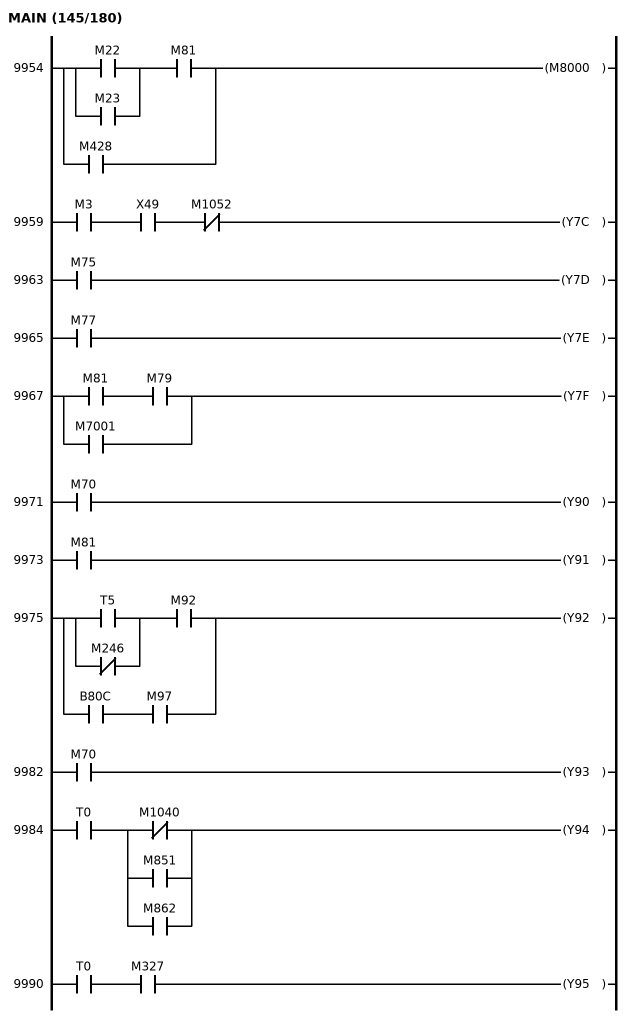
[picture p144: ladder of MAIN, rungs at steps 9954 to 9990]
9954  LD      M22
      OR      M23
      AND     M81
      OR      M428
      OUT     M8000
9959  LD      M3
      AND     X49
      ANI     M1052
      OUT     Y7C
9963  LD      M75
      OUT     Y7D
9965  LD      M77
      OUT     Y7E
9967  LD      M81
      AND     M79
      OR      M7001
      OUT     Y7F
9971  LD      M70
      OUT     Y90
9973  LD      M81
      OUT     Y91
9975  LD      T5
      ORI     M246
      AND     M92
      LD      B80C
      AND     M97
      ORB
      OUT     Y92
9982  LD      M70
      OUT     Y93
9984  LD      T0
      LDI     M1040
      OR      M851
      OR      M862
      ANB
      OUT     Y94
9990  LD      T0
      AND     M327
      OUT     Y95
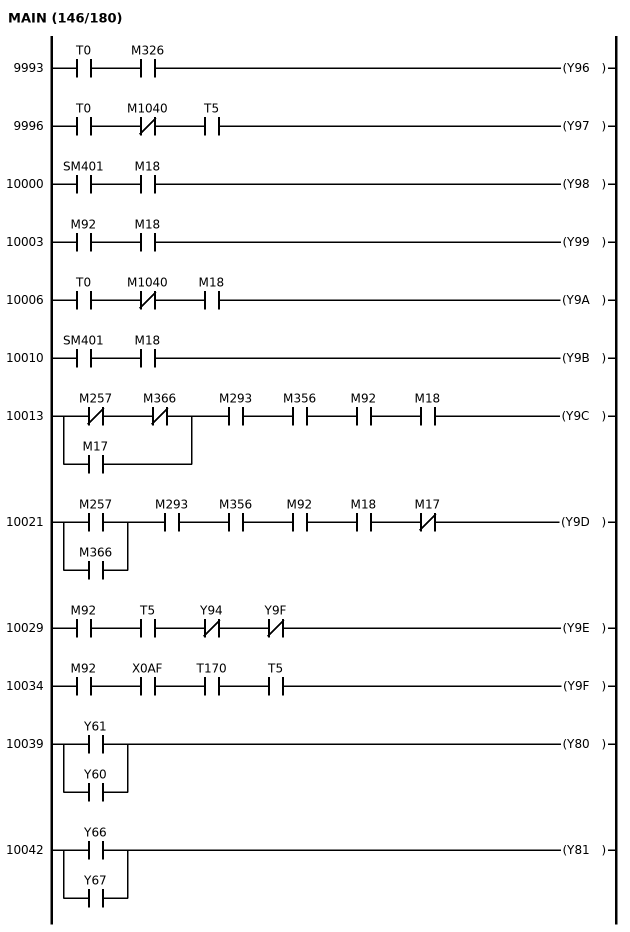
9993  LD      T0
      AND     M326
      OUT     Y96
9996  LD      T0
      ANI     M1040
      AND     T5
      OUT     Y97
10000 LD      SM401
      AND     M18
      OUT     Y98
10003 LD      M92
      AND     M18
      OUT     Y99
10006 LD      T0
      ANI     M1040
      AND     M18
      OUT     Y9A
10010 LD      SM401
      AND     M18
      OUT     Y9B
10013 LDI     M257
      ANI     M366
      OR      M17
      AND     M293
      AND     M356
      AND     M92
      AND     M18
      OUT     Y9C
10021 LD      M257
      OR      M366
      AND     M293
      AND     M356
      AND     M92
      AND     M18
      ANI     M17
      OUT     Y9D
10029 LD      M92
      AND     T5
      ANI     Y94
      ANI     Y9F
      OUT     Y9E
10034 LD      M92
      AND     X0AF
      AND     T170
      AND     T5
      OUT     Y9F
10039 LD      Y61
      OR      Y60
      OUT     Y80
10042 LD      Y66
      OR      Y67
      OUT     Y81
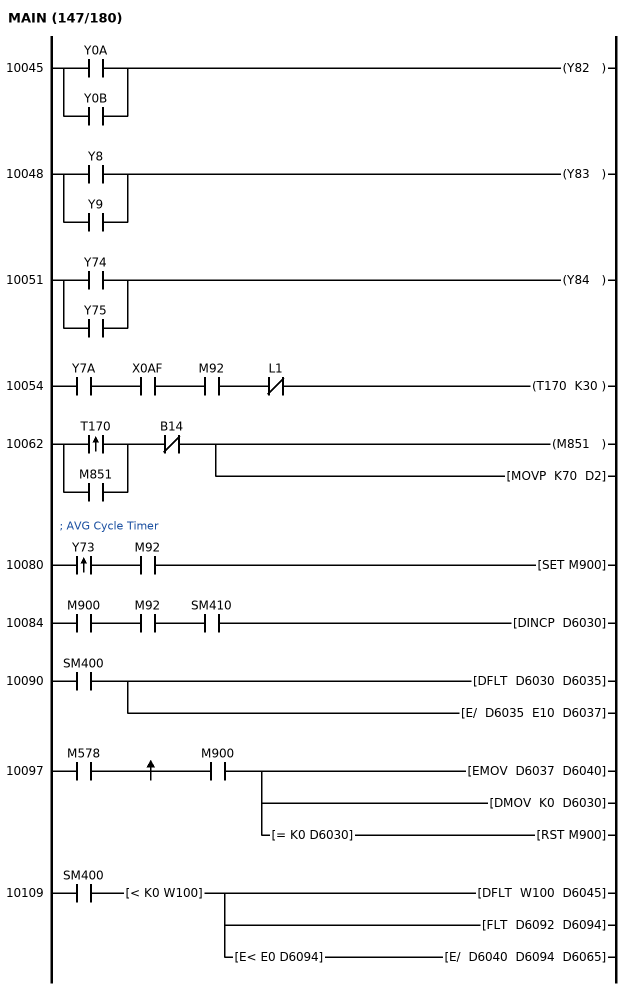
10045 LD      Y0A
      OR      Y0B
      OUT     Y82
10048 LD      Y8
      OR      Y9
      OUT     Y83
10051 LD      Y74
      OR      Y75
      OUT     Y84
10054 LD      Y7A
      AND     X0AF
      AND     M92
      ANI     L1
      OUT     T170 K30
10062 LDP     T170
      OR      M851
      ANI     B14
      OUT     M851
      MOVP    K70 D2
; AVG Cycle Timer
10080 LDP     Y73
      AND     M92
      SET     M900
10084 LD      M900
      AND     M92
      AND     SM410
      DINCP   D6030
10090 LD      SM400
      DFLT    D6030 D6035
      E/      D6035 E10 D6037
10097 LD      M578
      MEP
      AND     M900
      EMOV    D6037 D6040
      DMOV    K0 D6030
      AND=    K0 D6030
      RST     M900
10109 LD      SM400
      AND<    K0 W100
      DFLT    W100 D6045
      FLT     D6092 D6094
      ANDE<   E0 D6094
      E/      D6040 D6094 D6065
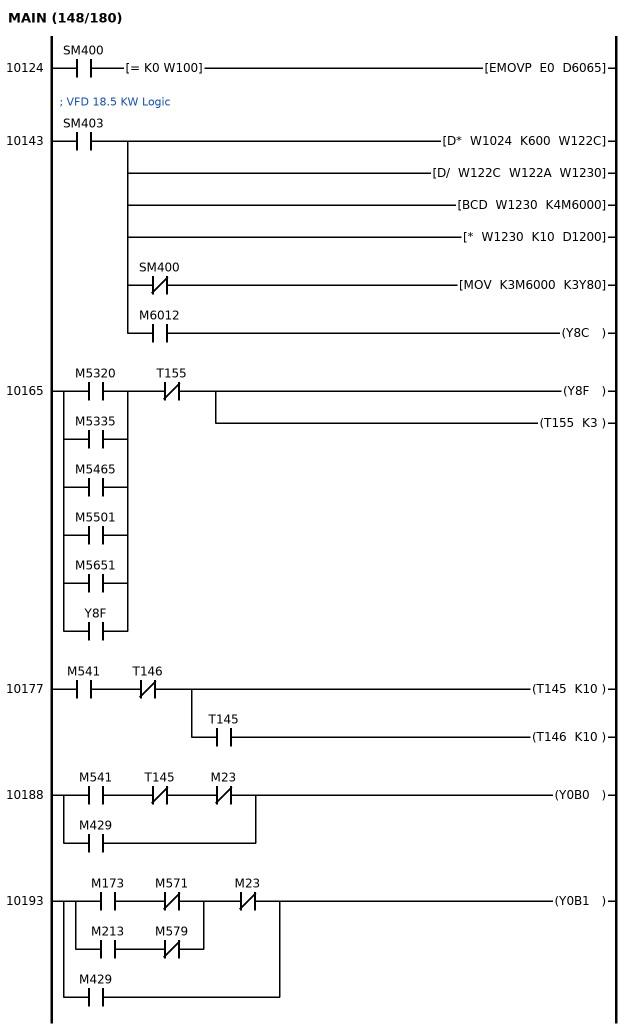
10124 LD      SM400
      AND=    K0 W100
      EMOVP   E0 D6065
; VFD 18.5 KW Logic
10143 LD      SM403
      D*      W1024 K600 W122C
      D/      W122C W122A W1230
      BCD     W1230 K4M6000
      *       W1230 K10 D1200
      MPS
      ANI     SM400
      MOV     K3M6000 K3Y80
      MPP
      AND     M6012
      OUT     Y8C
10165 LD      M5320
      OR      M5335
      OR      M5465
      OR      M5501
      OR      M5651
      OR      Y8F
      ANI     T155
      OUT     Y8F
      OUT     T155 K3
10177 LD      M541
      ANI     T146
      OUT     T145 K10
      AND     T145
      OUT     T146 K10
10188 LD      M541
      ANI     T145
      ANI     M23
      OR      M429
      OUT     Y0B0
10193 LD      M173
      ANI     M571
      LD      M213
      ANI     M579
      ORB
      ANI     M23
      OR      M429
      OUT     Y0B1
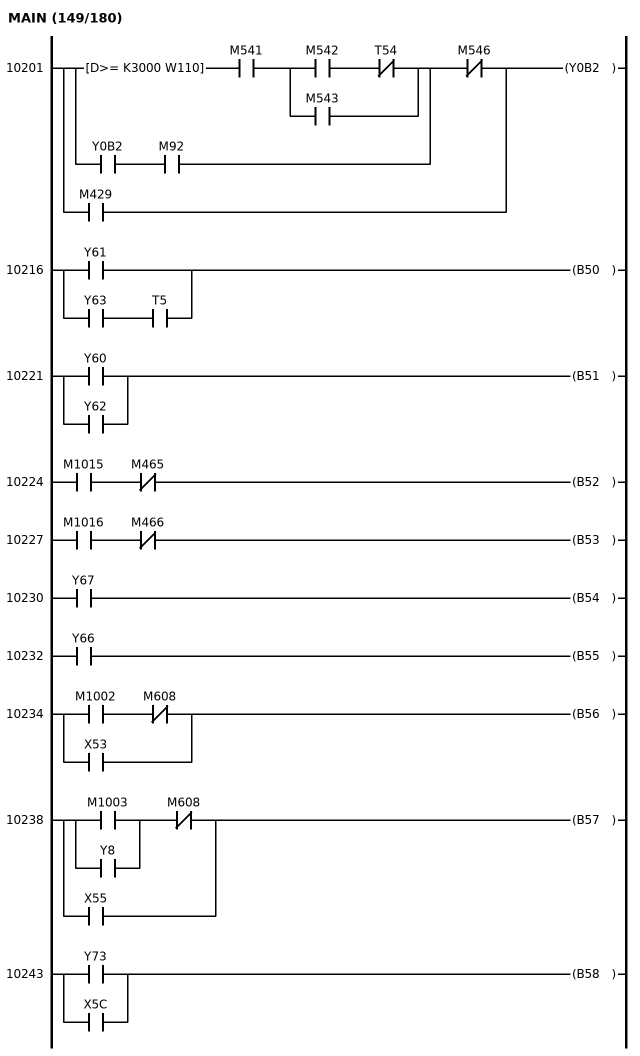
10201 LDD>=   K3000 W110
      AND     M541
      LD      M542
      ANI     T54
      OR      M543
      ANB
      LD      Y0B2
      AND     M92
      ORB
      ANI     M546
      OR      M429
      OUT     Y0B2
10216 LD      Y61
      LD      Y63
      AND     T5
      ORB
      OUT     B50
10221 LD      Y60
      OR      Y62
      OUT     B51
10224 LD      M1015
      ANI     M465
      OUT     B52
10227 LD      M1016
      ANI     M466
      OUT     B53
10230 LD      Y67
      OUT     B54
10232 LD      Y66
      OUT     B55
10234 LD      M1002
      ANI     M608
      OR      X53
      OUT     B56
10238 LD      M1003
      OR      Y8
      ANI     M608
      OR      X55
      OUT     B57
10243 LD      Y73
      OR      X5C
      OUT     B58
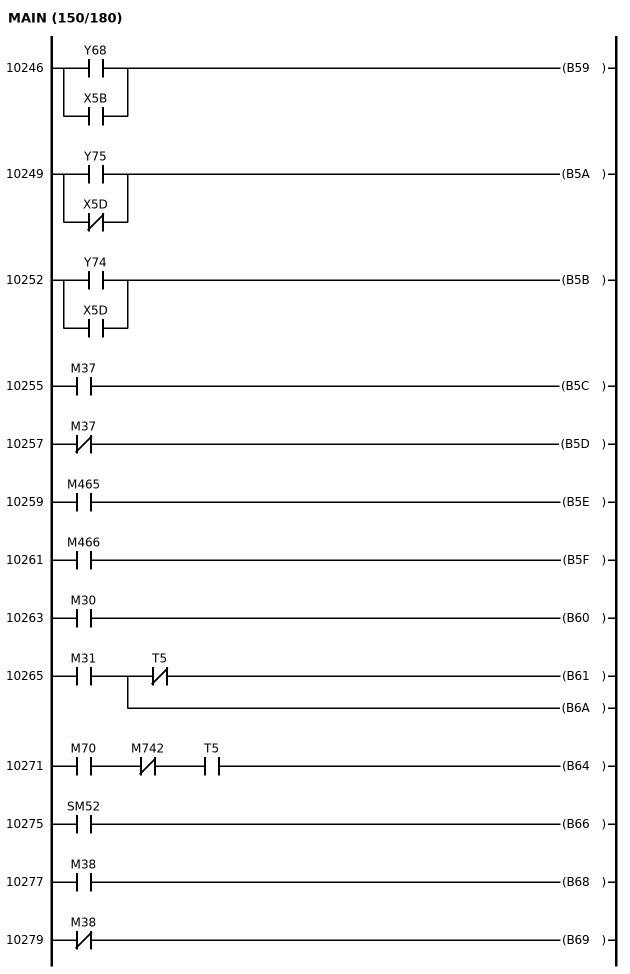
10246 LD      Y68
      OR      X5B
      OUT     B59
10249 LD      Y75
      ORI     X5D
      OUT     B5A
10252 LD      Y74
      OR      X5D
      OUT     B5B
10255 LD      M37
      OUT     B5C
10257 LDI     M37
      OUT     B5D
10259 LD      M465
      OUT     B5E
10261 LD      M466
      OUT     B5F
10263 LD      M30
      OUT     B60
10265 LD      M31
      MPS
      ANI     T5
      OUT     B61
      MPP
      OUT     B6A
10271 LD      M70
      ANI     M742
      AND     T5
      OUT     B64
10275 LD      SM52
      OUT     B66
10277 LD      M38
      OUT     B68
10279 LDI     M38
      OUT     B69
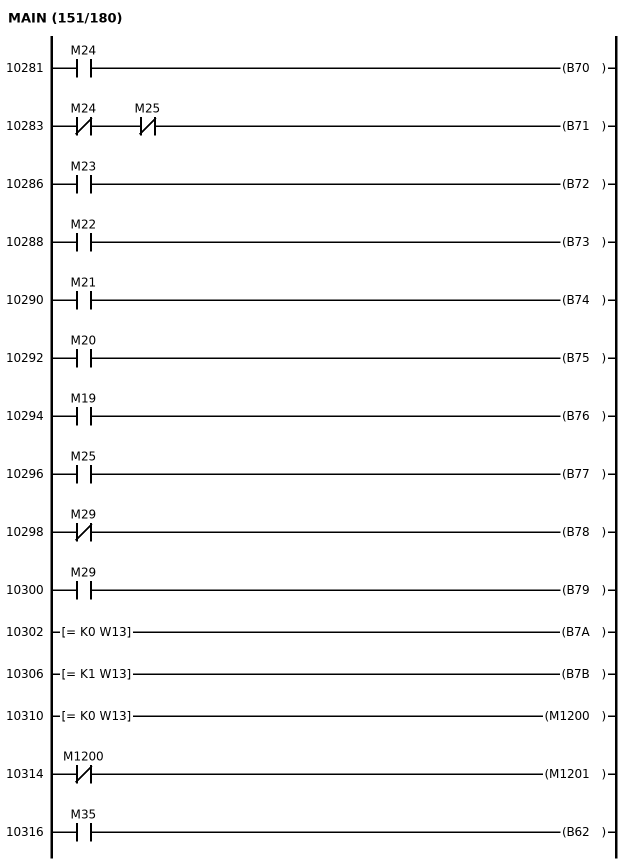
10281 LD      M24
      OUT     B70
10283 LDI     M24
      ANI     M25
      OUT     B71
10286 LD      M23
      OUT     B72
10288 LD      M22
      OUT     B73
10290 LD      M21
      OUT     B74
10292 LD      M20
      OUT     B75
10294 LD      M19
      OUT     B76
10296 LD      M25
      OUT     B77
10298 LDI     M29
      OUT     B78
10300 LD      M29
      OUT     B79
10302 LD=     K0 W13
      OUT     B7A
10306 LD=     K1 W13
      OUT     B7B
10310 LD=     K0 W13
      OUT     M1200
10314 LDI     M1200
      OUT     M1201
10316 LD      M35
      OUT     B62
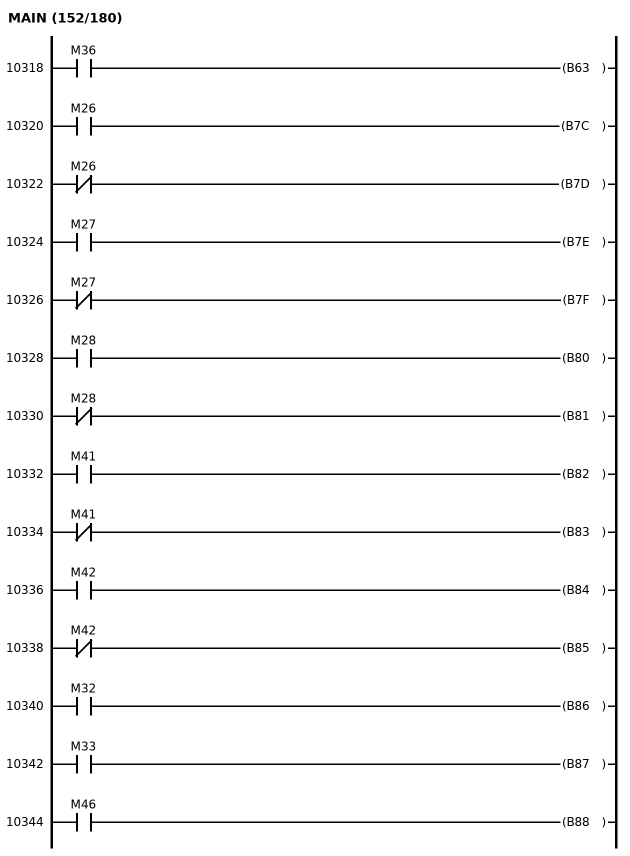
10318 LD      M36
      OUT     B63
10320 LD      M26
      OUT     B7C
10322 LDI     M26
      OUT     B7D
10324 LD      M27
      OUT     B7E
10326 LDI     M27
      OUT     B7F
10328 LD      M28
      OUT     B80
10330 LDI     M28
      OUT     B81
10332 LD      M41
      OUT     B82
10334 LDI     M41
      OUT     B83
10336 LD      M42
      OUT     B84
10338 LDI     M42
      OUT     B85
10340 LD      M32
      OUT     B86
10342 LD      M33
      OUT     B87
10344 LD      M46
      OUT     B88
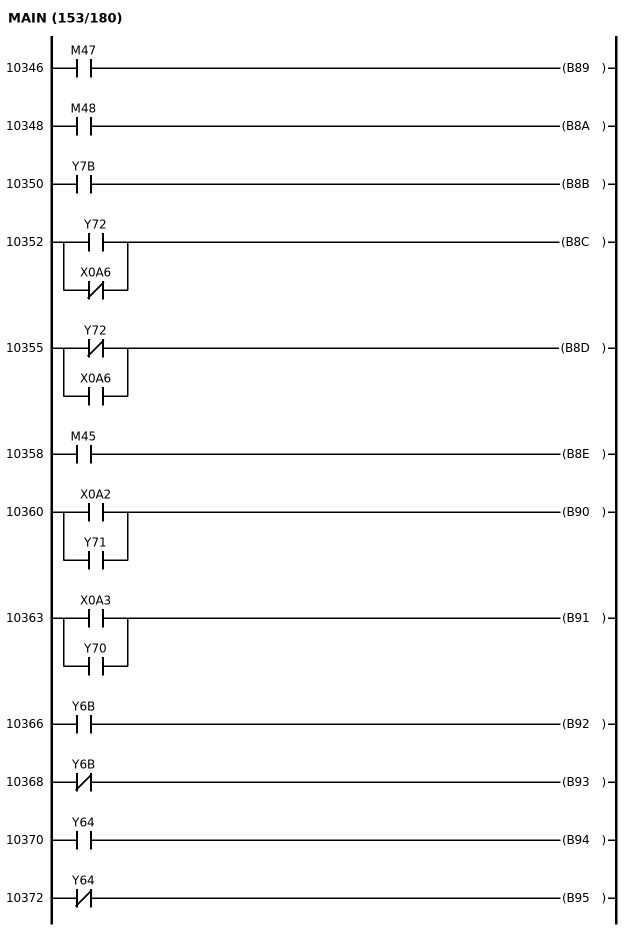
10346 LD      M47
      OUT     B89
10348 LD      M48
      OUT     B8A
10350 LD      Y7B
      OUT     B8B
10352 LD      Y72
      ORI     X0A6
      OUT     B8C
10355 LDI     Y72
      OR      X0A6
      OUT     B8D
10358 LD      M45
      OUT     B8E
10360 LD      X0A2
      OR      Y71
      OUT     B90
10363 LD      X0A3
      OR      Y70
      OUT     B91
10366 LD      Y6B
      OUT     B92
10368 LDI     Y6B
      OUT     B93
10370 LD      Y64
      OUT     B94
10372 LDI     Y64
      OUT     B95
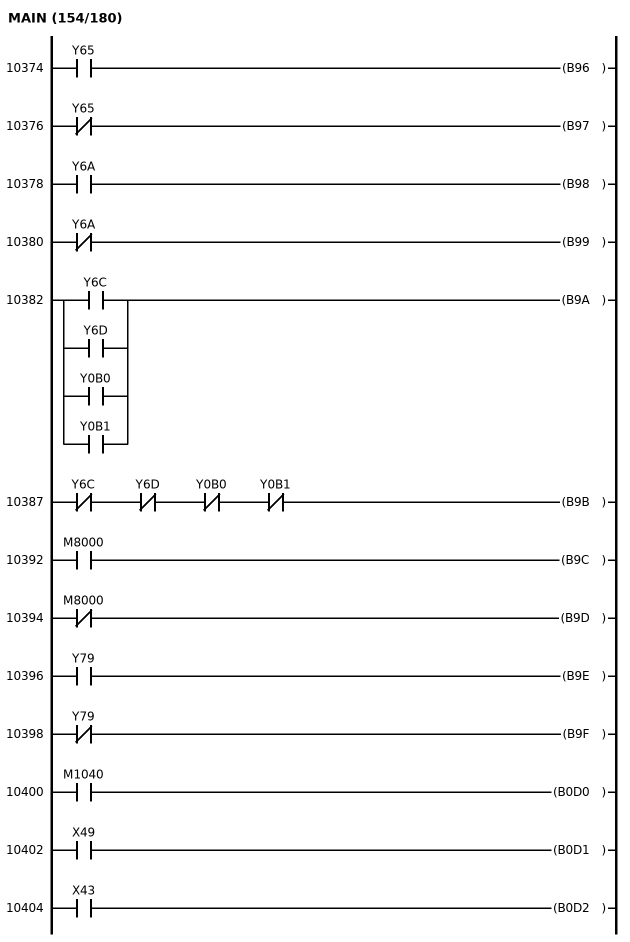
10374 LD      Y65
      OUT     B96
10376 LDI     Y65
      OUT     B97
10378 LD      Y6A
      OUT     B98
10380 LDI     Y6A
      OUT     B99
10382 LD      Y6C
      OR      Y6D
      OR      Y0B0
      OR      Y0B1
      OUT     B9A
10387 LDI     Y6C
      ANI     Y6D
      ANI     Y0B0
      ANI     Y0B1
      OUT     B9B
10392 LD      M8000
      OUT     B9C
10394 LDI     M8000
      OUT     B9D
10396 LD      Y79
      OUT     B9E
10398 LDI     Y79
      OUT     B9F
10400 LD      M1040
      OUT     B0D0
10402 LD      X49
      OUT     B0D1
10404 LD      X43
      OUT     B0D2
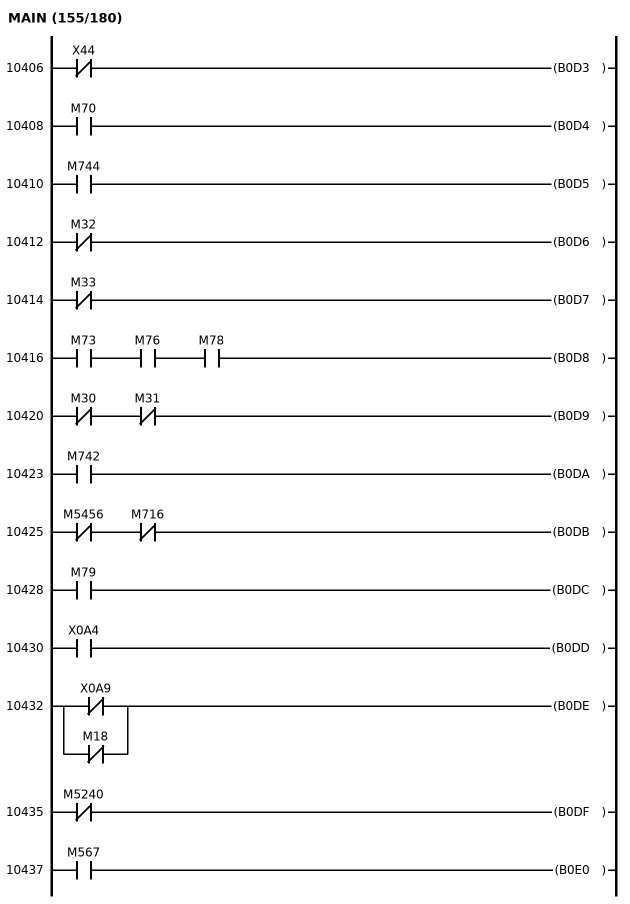
10406 LDI     X44
      OUT     B0D3
10408 LD      M70
      OUT     B0D4
10410 LD      M744
      OUT     B0D5
10412 LDI     M32
      OUT     B0D6
10414 LDI     M33
      OUT     B0D7
10416 LD      M73
      AND     M76
      AND     M78
      OUT     B0D8
10420 LDI     M30
      ANI     M31
      OUT     B0D9
10423 LD      M742
      OUT     B0DA
10425 LDI     M5456
      ANI     M716
      OUT     B0DB
10428 LD      M79
      OUT     B0DC
10430 LD      X0A4
      OUT     B0DD
10432 LDI     X0A9
      ORI     M18
      OUT     B0DE
10435 LDI     M5240
      OUT     B0DF
10437 LD      M567
      OUT     B0E0
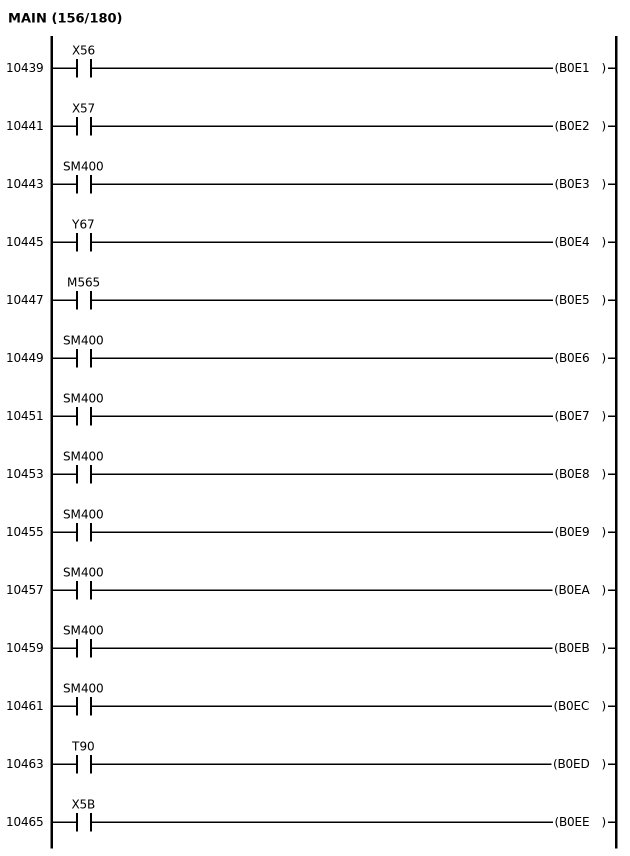
10439 LD      X56
      OUT     B0E1
10441 LD      X57
      OUT     B0E2
10443 LD      SM400
      OUT     B0E3
10445 LD      Y67
      OUT     B0E4
10447 LD      M565
      OUT     B0E5
10449 LD      SM400
      OUT     B0E6
10451 LD      SM400
      OUT     B0E7
10453 LD      SM400
      OUT     B0E8
10455 LD      SM400
      OUT     B0E9
10457 LD      SM400
      OUT     B0EA
10459 LD      SM400
      OUT     B0EB
10461 LD      SM400
      OUT     B0EC
10463 LD      T90
      OUT     B0ED
10465 LD      X5B
      OUT     B0EE
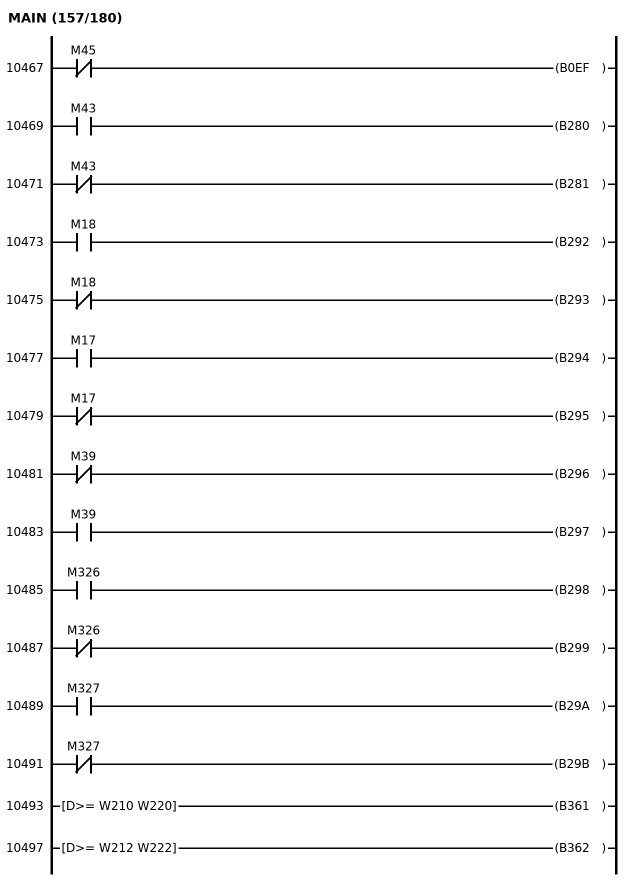
10467 LDI     M45
      OUT     B0EF
10469 LD      M43
      OUT     B280
10471 LDI     M43
      OUT     B281
10473 LD      M18
      OUT     B292
10475 LDI     M18
      OUT     B293
10477 LD      M17
      OUT     B294
10479 LDI     M17
      OUT     B295
10481 LDI     M39
      OUT     B296
10483 LD      M39
      OUT     B297
10485 LD      M326
      OUT     B298
10487 LDI     M326
      OUT     B299
10489 LD      M327
      OUT     B29A
10491 LDI     M327
      OUT     B29B
10493 LDD>=   W210 W220
      OUT     B361
10497 LDD>=   W212 W222
      OUT     B362
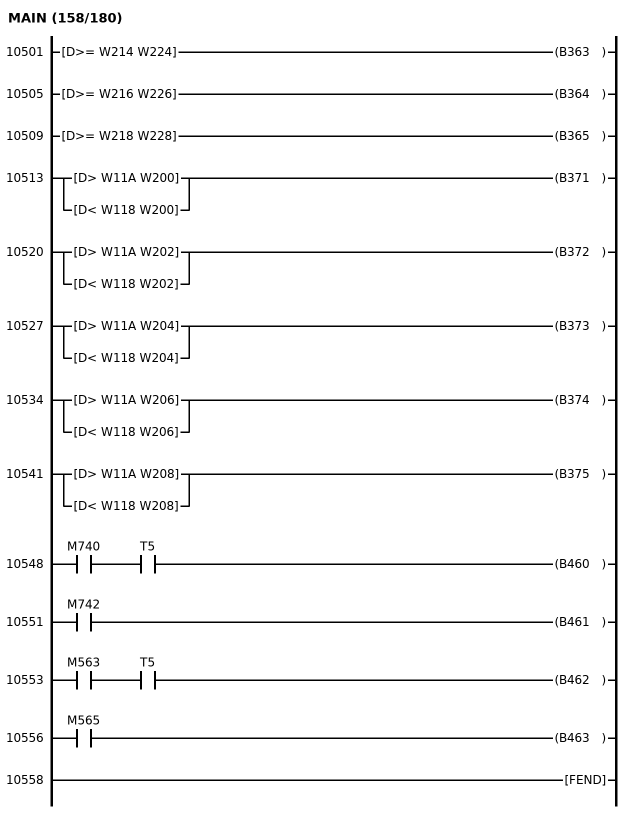
10501 LDD>=   W214 W224
      OUT     B363
10505 LDD>=   W216 W226
      OUT     B364
10509 LDD>=   W218 W228
      OUT     B365
10513 LDD>    W11A W200
      ORD<    W118 W200
      OUT     B371
10520 LDD>    W11A W202
      ORD<    W118 W202
      OUT     B372
10527 LDD>    W11A W204
      ORD<    W118 W204
      OUT     B373
10534 LDD>    W11A W206
      ORD<    W118 W206
      OUT     B374
10541 LDD>    W11A W208
      ORD<    W118 W208
      OUT     B375
10548 LD      M740
      AND     T5
      OUT     B460
10551 LD      M742
      OUT     B461
10553 LD      M563
      AND     T5
      OUT     B462
10556 LD      M565
      OUT     B463
10558 FEND
      P0
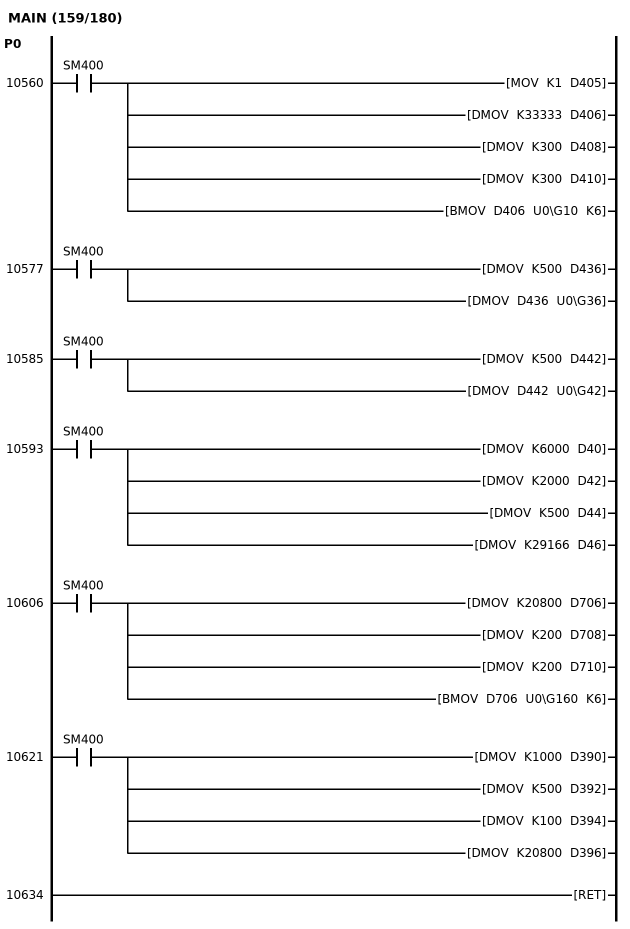
10560 LD      SM400
      MOV     K1 D405
      DMOV    K33333 D406
      DMOV    K300 D408
      DMOV    K300 D410
      BMOV    D406 U0\G10 K6
10577 LD      SM400
      DMOV    K500 D436
      DMOV    D436 U0\G36
10585 LD      SM400
      DMOV    K500 D442
      DMOV    D442 U0\G42
10593 LD      SM400
      DMOV    K6000 D40
      DMOV    K2000 D42
      DMOV    K500 D44
      DMOV    K29166 D46
10606 LD      SM400
      DMOV    K20800 D706
      DMOV    K200 D708
      DMOV    K200 D710
      BMOV    D706 U0\G160 K6
10621 LD      SM400
      DMOV    K1000 D390
      DMOV    K500 D392
      DMOV    K100 D394
      DMOV    K20800 D396
10634 RET
      P1
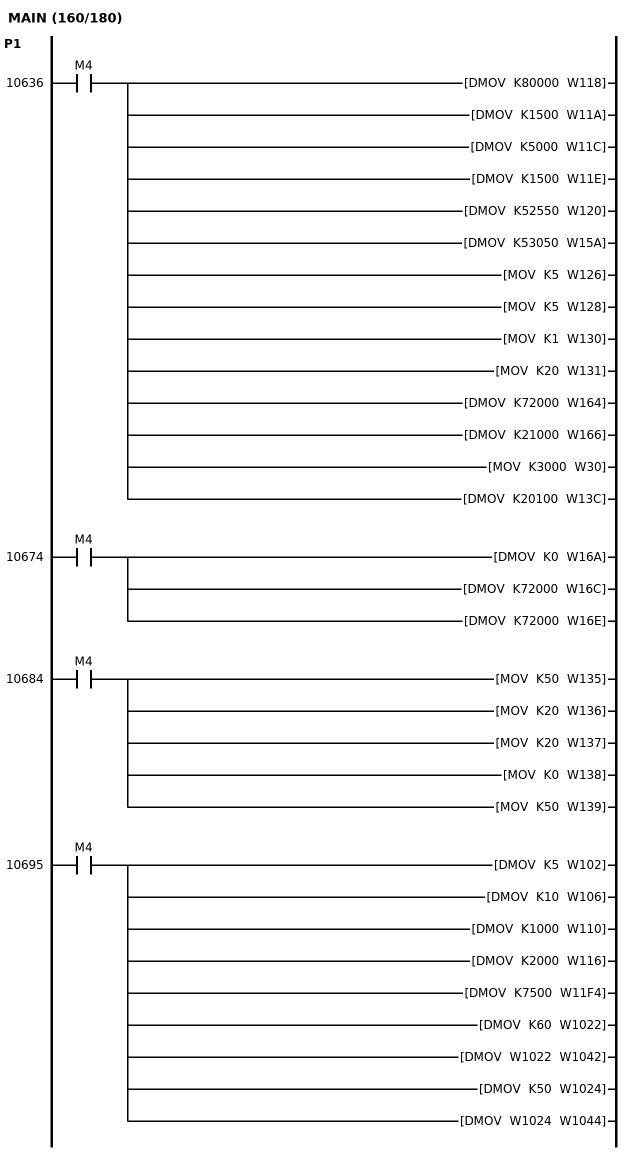
10636 LD      M4
      DMOV    K80000 W118
      DMOV    K1500 W11A
      DMOV    K5000 W11C
      DMOV    K1500 W11E
      DMOV    K52550 W120
      DMOV    K53050 W15A
      MOV     K5 W126
      MOV     K5 W128
      MOV     K1 W130
      MOV     K20 W131
      DMOV    K72000 W164
      DMOV    K21000 W166
      MOV     K3000 W30
      DMOV    K20100 W13C
10674 LD      M4
      DMOV    K0 W16A
      DMOV    K72000 W16C
      DMOV    K72000 W16E
10684 LD      M4
      MOV     K50 W135
      MOV     K20 W136
      MOV     K20 W137
      MOV     K0 W138
      MOV     K50 W139
10695 LD      M4
      DMOV    K5 W102
      DMOV    K10 W106
      DMOV    K1000 W110
      DMOV    K2000 W116
      DMOV    K7500 W11F4
      DMOV    K60 W1022
      DMOV    W1022 W1042
      DMOV    K50 W1024
      DMOV    W1024 W1044
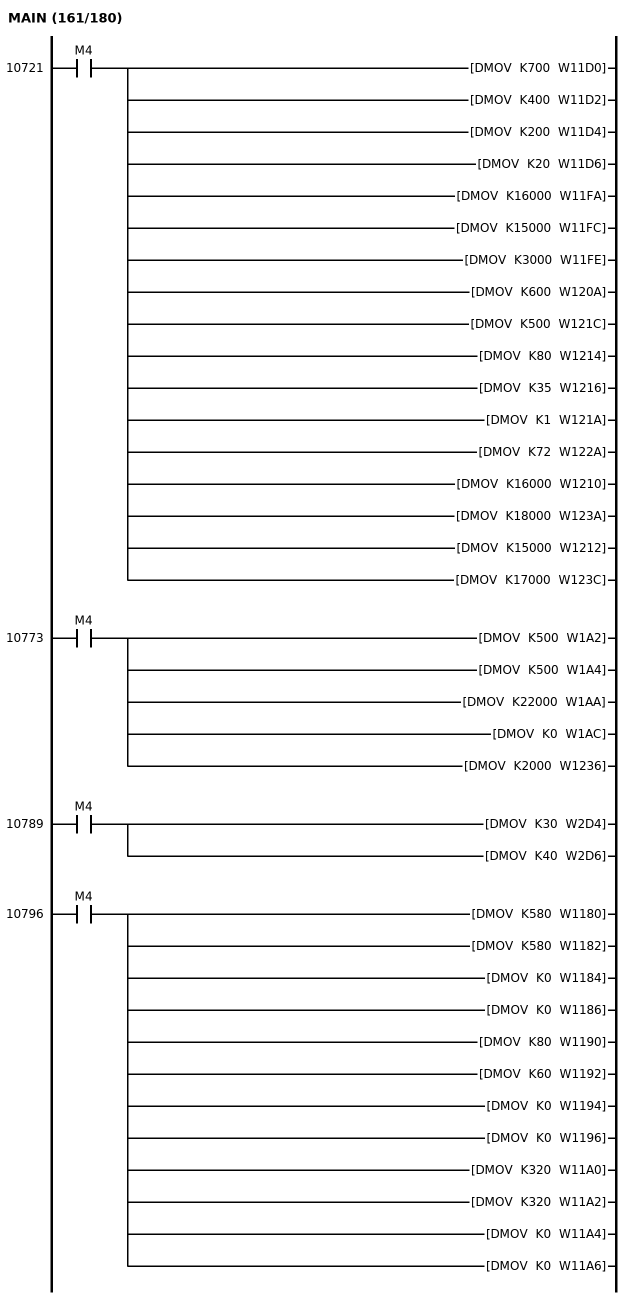
10721 LD      M4
      DMOV    K700 W11D0
      DMOV    K400 W11D2
      DMOV    K200 W11D4
      DMOV    K20 W11D6
      DMOV    K16000 W11FA
      DMOV    K15000 W11FC
      DMOV    K3000 W11FE
      DMOV    K600 W120A
      DMOV    K500 W121C
      DMOV    K80 W1214
      DMOV    K35 W1216
      DMOV    K1 W121A
      DMOV    K72 W122A
      DMOV    K16000 W1210
      DMOV    K18000 W123A
      DMOV    K15000 W1212
      DMOV    K17000 W123C
10773 LD      M4
      DMOV    K500 W1A2
      DMOV    K500 W1A4
      DMOV    K22000 W1AA
      DMOV    K0 W1AC
      DMOV    K2000 W1236
10789 LD      M4
      DMOV    K30 W2D4
      DMOV    K40 W2D6
10796 LD      M4
      DMOV    K580 W1180
      DMOV    K580 W1182
      DMOV    K0 W1184
      DMOV    K0 W1186
      DMOV    K80 W1190
      DMOV    K60 W1192
      DMOV    K0 W1194
      DMOV    K0 W1196
      DMOV    K320 W11A0
      DMOV    K320 W11A2
      DMOV    K0 W11A4
      DMOV    K0 W11A6
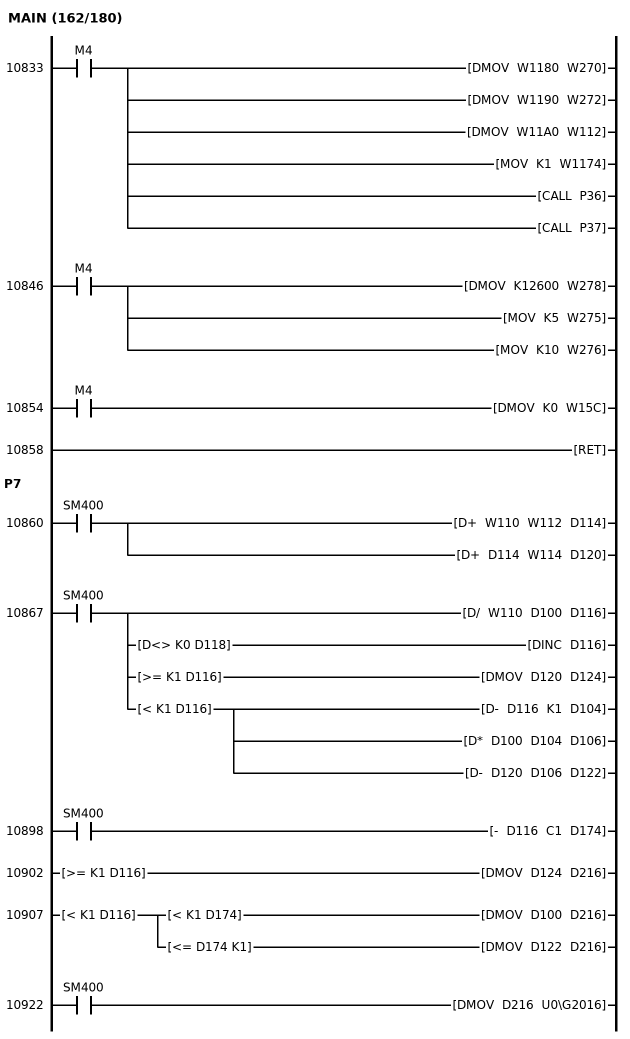
10833 LD      M4
      DMOV    W1180 W270
      DMOV    W1190 W272
      DMOV    W11A0 W112
      MOV     K1 W1174
      CALL    P36
      CALL    P37
10846 LD      M4
      DMOV    K12600 W278
      MOV     K5 W275
      MOV     K10 W276
10854 LD      M4
      DMOV    K0 W15C
10858 RET
      P7
10860 LD      SM400
      D+      W110 W112 D114
      D+      D114 W114 D120
10867 LD      SM400
      D/      W110 D100 D116
      MPS
      ANDD<>  K0 D118
      DINC    D116
      MRD
      AND>=   K1 D116
      DMOV    D120 D124
      MPP
      AND<    K1 D116
      D-      D116 K1 D104
      D*      D100 D104 D106
      D-      D120 D106 D122
10898 LD      SM400
      -       D116 C1 D174
10902 LD>=    K1 D116
      DMOV    D124 D216
10907 LD<     K1 D116
      MPS
      AND<    K1 D174
      DMOV    D100 D216
      MPP
      AND<=   D174 K1
      DMOV    D122 D216
10922 LD      SM400
      DMOV    D216 U0\G2016
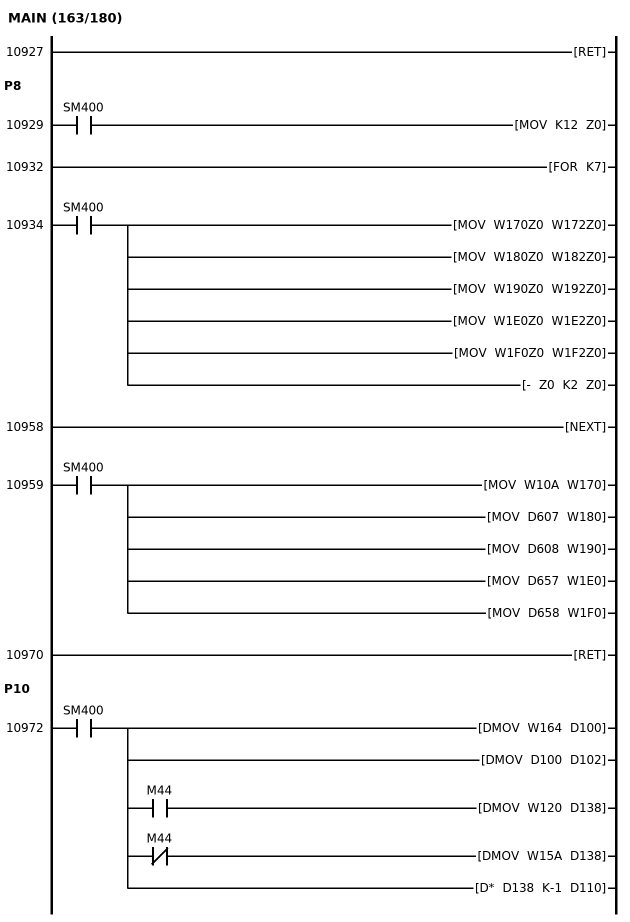
10927 RET
      P8
10929 LD      SM400
      MOV     K12 Z0
10932 FOR     K7
10934 LD      SM400
      MOV     W170Z0 W172Z0
      MOV     W180Z0 W182Z0
      MOV     W190Z0 W192Z0
      MOV     W1E0Z0 W1E2Z0
      MOV     W1F0Z0 W1F2Z0
      -       Z0 K2 Z0
10958 NEXT
10959 LD      SM400
      MOV     W10A W170
      MOV     D607 W180
      MOV     D608 W190
      MOV     D657 W1E0
      MOV     D658 W1F0
10970 RET
      P10
10972 LD      SM400
      DMOV    W164 D100
      DMOV    D100 D102
      MPS
      AND     M44
      DMOV    W120 D138
      MRD
      ANI     M44
      DMOV    W15A D138
      MPP
      D*      D138 K-1 D110
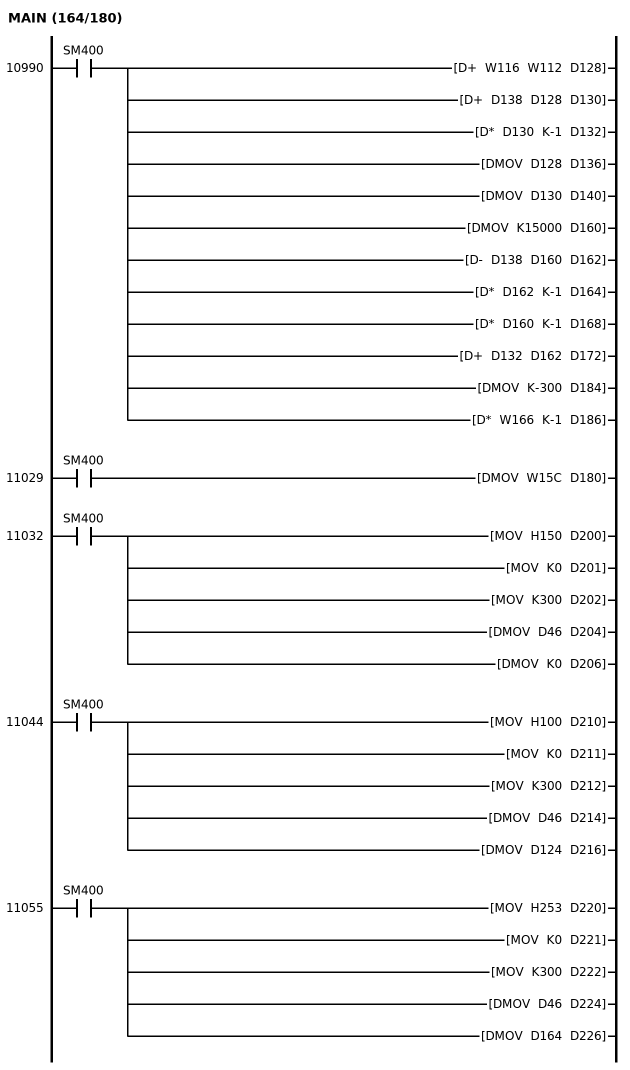
10990 LD      SM400
      D+      W116 W112 D128
      D+      D138 D128 D130
      D*      D130 K-1 D132
      DMOV    D128 D136
      DMOV    D130 D140
      DMOV    K15000 D160
      D-      D138 D160 D162
      D*      D162 K-1 D164
      D*      D160 K-1 D168
      D+      D132 D162 D172
      DMOV    K-300 D184
      D*      W166 K-1 D186
11029 LD      SM400
      DMOV    W15C D180
11032 LD      SM400
      MOV     H150 D200
      MOV     K0 D201
      MOV     K300 D202
      DMOV    D46 D204
      DMOV    K0 D206
11044 LD      SM400
      MOV     H100 D210
      MOV     K0 D211
      MOV     K300 D212
      DMOV    D46 D214
      DMOV    D124 D216
11055 LD      SM400
      MOV     H253 D220
      MOV     K0 D221
      MOV     K300 D222
      DMOV    D46 D224
      DMOV    D164 D226
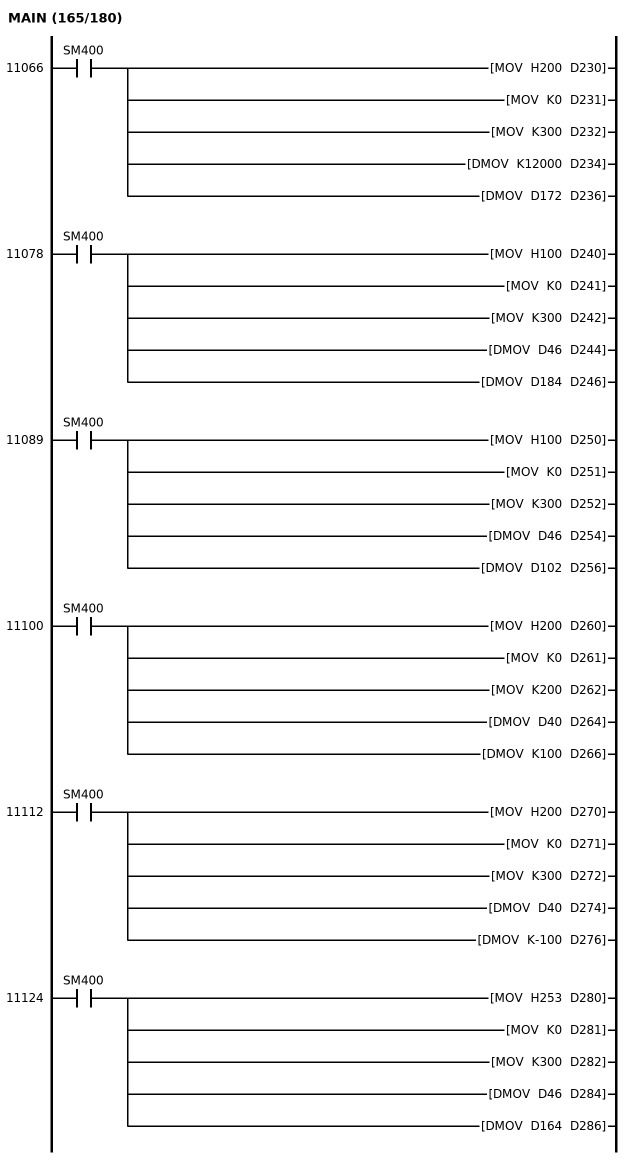
11066 LD      SM400
      MOV     H200 D230
      MOV     K0 D231
      MOV     K300 D232
      DMOV    K12000 D234
      DMOV    D172 D236
11078 LD      SM400
      MOV     H100 D240
      MOV     K0 D241
      MOV     K300 D242
      DMOV    D46 D244
      DMOV    D184 D246
11089 LD      SM400
      MOV     H100 D250
      MOV     K0 D251
      MOV     K300 D252
      DMOV    D46 D254
      DMOV    D102 D256
11100 LD      SM400
      MOV     H200 D260
      MOV     K0 D261
      MOV     K200 D262
      DMOV    D40 D264
      DMOV    K100 D266
11112 LD      SM400
      MOV     H200 D270
      MOV     K0 D271
      MOV     K300 D272
      DMOV    D40 D274
      DMOV    K-100 D276
11124 LD      SM400
      MOV     H253 D280
      MOV     K0 D281
      MOV     K300 D282
      DMOV    D46 D284
      DMOV    D164 D286
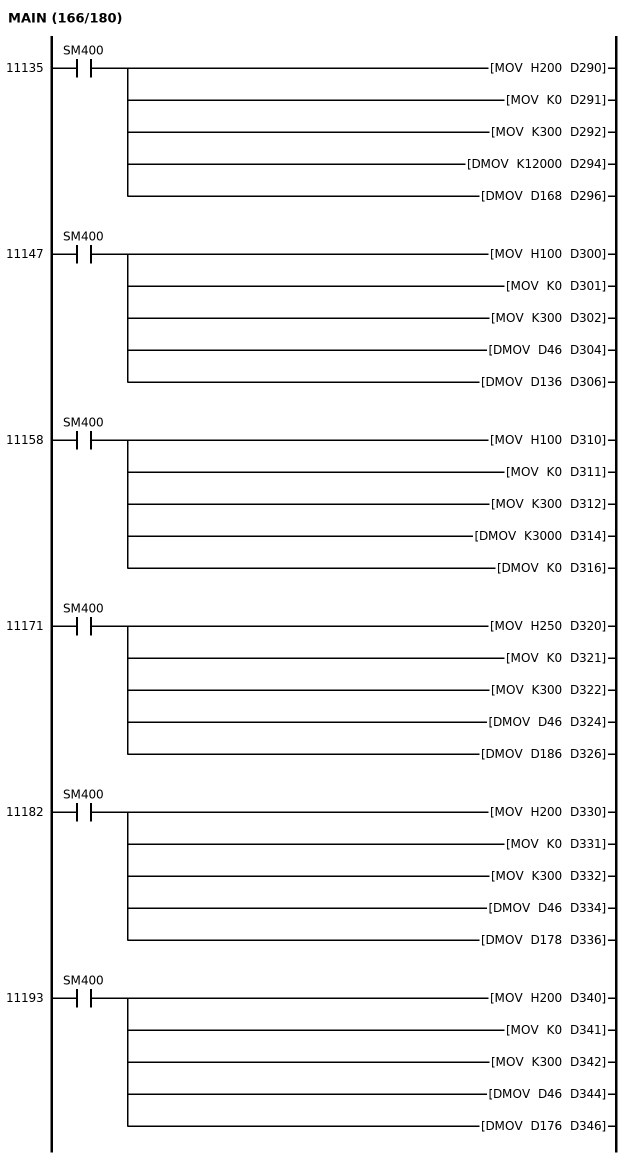
11135 LD      SM400
      MOV     H200 D290
      MOV     K0 D291
      MOV     K300 D292
      DMOV    K12000 D294
      DMOV    D168 D296
11147 LD      SM400
      MOV     H100 D300
      MOV     K0 D301
      MOV     K300 D302
      DMOV    D46 D304
      DMOV    D136 D306
11158 LD      SM400
      MOV     H100 D310
      MOV     K0 D311
      MOV     K300 D312
      DMOV    K3000 D314
      DMOV    K0 D316
11171 LD      SM400
      MOV     H250 D320
      MOV     K0 D321
      MOV     K300 D322
      DMOV    D46 D324
      DMOV    D186 D326
11182 LD      SM400
      MOV     H200 D330
      MOV     K0 D331
      MOV     K300 D332
      DMOV    D46 D334
      DMOV    D178 D336
11193 LD      SM400
      MOV     H200 D340
      MOV     K0 D341
      MOV     K300 D342
      DMOV    D46 D344
      DMOV    D176 D346
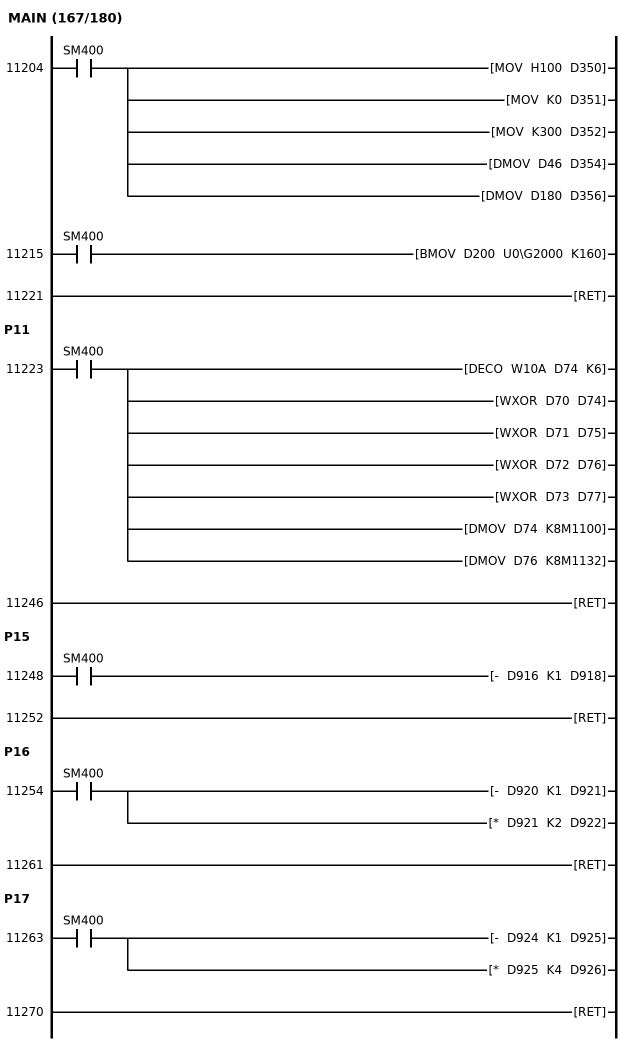
11204 LD      SM400
      MOV     H100 D350
      MOV     K0 D351
      MOV     K300 D352
      DMOV    D46 D354
      DMOV    D180 D356
11215 LD      SM400
      BMOV    D200 U0\G2000 K160
11221 RET
      P11
11223 LD      SM400
      DECO    W10A D74 K6
      WXOR    D70 D74
      WXOR    D71 D75
      WXOR    D72 D76
      WXOR    D73 D77
      DMOV    D74 K8M1100
      DMOV    D76 K8M1132
11246 RET
      P15
11248 LD      SM400
      -       D916 K1 D918
11252 RET
      P16
11254 LD      SM400
      -       D920 K1 D921
      *       D921 K2 D922
11261 RET
      P17
11263 LD      SM400
      -       D924 K1 D925
      *       D925 K4 D926
11270 RET
      P21
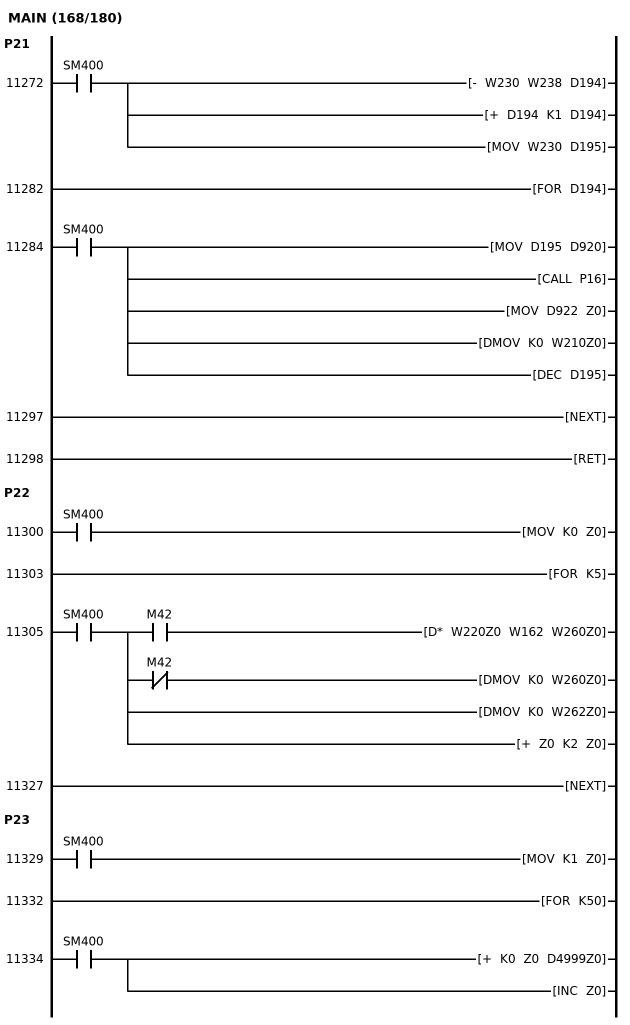
11272 LD      SM400
      -       W230 W238 D194
      +       D194 K1 D194
      MOV     W230 D195
11282 FOR     D194
11284 LD      SM400
      MOV     D195 D920
      CALL    P16
      MOV     D922 Z0
      DMOV    K0 W210Z0
      DEC     D195
11297 NEXT
11298 RET
      P22
11300 LD      SM400
      MOV     K0 Z0
11303 FOR     K5
11305 LD      SM400
      MPS
      AND     M42
      D*      W220Z0 W162 W260Z0
      MRD
      ANI     M42
      DMOV    K0 W260Z0
      MPP
      DMOV    K0 W262Z0
      +       Z0 K2 Z0
11327 NEXT
      P23
11329 LD      SM400
      MOV     K1 Z0
11332 FOR     K50
11334 LD      SM400
      +       K0 Z0 D4999Z0
      INC     Z0
